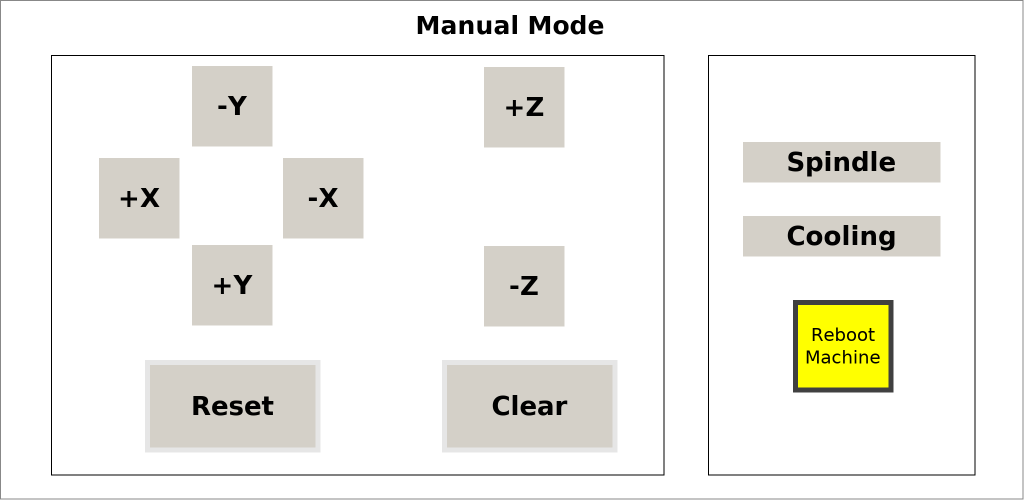
VISUALIZATION V_ManualMode  // 1024x500
VAR_IN_OUT
	HMI : ST_PackMLBaseModule_HMI;
	HMIAxeX : ST_AxisBase_HMI;
	HMIAxeY : ST_AxisBase_HMI;
	HMIAxeZ : ST_AxisBase_HMI;
END_VAR
    RoundedRectangle (51,55 613x420)
    RoundedRectangle (708,55 267x420)
    Label (0,0 1020x50), "Manual Mode"
    RoundedRectangle (738,137 207x50), "Spindle", colour toggle: HMI.Status.State = E_PMLState.ePMLState_Idle
        toggle SpindleEnable
    RoundedRectangle (738,211 207x50), "Cooling", colour toggle: HMI.Status.State = E_PMLState.ePMLState_Idle
        toggle CoolingEnable
    RoundedRectangle (283,158 80x80), "-X", colour toggle: HMI.Status.State = E_PMLState.ePMLState_Idle
        tap HMIAxeX.Command.JogFast_Backward
        OnMouseClick: execute { HMI.Command.State := E_PMLCommand.ePMLCommand_Clear; }
    RoundedRectangle (99,158 80x80), "+X", colour toggle: HMI.Status.State = E_PMLState.ePMLState_Idle
        tap HMIAxeX.Command.JogFast_Forward
    RoundedRectangle (192,245 80x80), "+Y", colour toggle: HMI.Status.State = E_PMLState.ePMLState_Idle
        tap HMIAxeY.Command.JogFast_Forward
    RoundedRectangle (192,66 80x80), "-Y", colour toggle: HMI.Status.State = E_PMLState.ePMLState_Idle
        tap HMIAxeY.Command.JogFast_Backward
        OnMouseClick: execute { HMI.Command.State := E_PMLCommand.ePMLCommand_Clear; }
    RoundedRectangle (484,67 80x80), "+Z", colour toggle: HMI.Status.State = E_PMLState.ePMLState_Idle
        tap HMIAxeZ.Command.JogSlow_Forward
    RoundedRectangle (484,246 80x80), "-Z", colour toggle: HMI.Status.State = E_PMLState.ePMLState_Idle
        tap HMIAxeZ.Command.JogSlow_Backward p3779583253=TRUE
    Rectangle (793,300 100x92), "Reboot Machine"
        OnMouseClick: execute { MAIN.RebootSystem(DELAY:=5,START:=TRUE); }
    RoundedRectangle (442,360 175x92), "Clear", colour toggle: (HMI.Status.State = E_PMLState.ePMLState_Aborted) OR (HMI.Status.State = E_PMLState.ePMLState_Clearing)
        OnMouseClick: execute { HMI.Command.State := E_PMLCommand.ePMLCommand_Clear; }
    RoundedRectangle (145,360 175x92), "Reset", colour toggle: (HMI.Status.State = E_PMLState.ePMLState_Complete) OR (HMI.Status.State = E_PMLState.ePMLState_Stopped) OR (HMI.Status.State = E_PMLState.ePMLState_Resetting)
        OnMouseClick: execute { HMI.Command.State := E_PMLCommand.ePMLCommand_Reset; }
END_VISUALIZATION

(* stored: Version 1.1.0.1, ProductVersion 3.1.4024.15
   Visu V_ManualMode: Id {5eb24302-7c74-4cb0-913c-af4cad05dac4} *)
